PROGRAM pouS1Alarms
VAR
	idbMsgAlarm: FB_CheckMessageBounds;

END_VAR

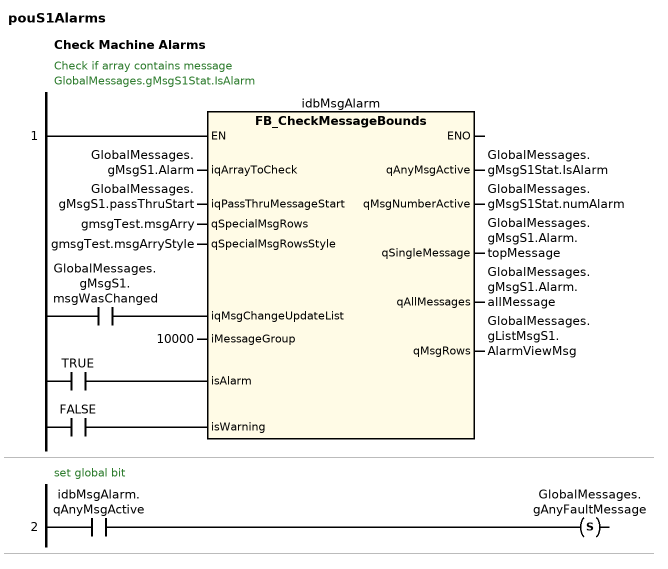
// NETWORK 1: Check Machine Alarms
// Check if array contains message
//
// GlobalMessages.gMsgS1Stat.IsAlarm
idbMsgAlarm(
    iqArrayToCheck := GlobalMessages.gMsgS1.Alarm,
    iqPassThruMessageStart := GlobalMessages.gMsgS1.passThruStart,
    qSpecialMsgRows := gmsgTest.msgArry,
    qSpecialMsgRowsStyle := gmsgTest.msgArryStyle,
    iqMsgChangeUpdateList := GlobalMessages.gMsgS1.msgWasChanged,
    iMessageGroup := 10000,
    isAlarm := TRUE,
    isWarning := FALSE,
    qAnyMsgActive => GlobalMessages.gMsgS1Stat.IsAlarm,
    qMsgNumberActive => GlobalMessages.gMsgS1Stat.numAlarm,
    qSingleMessage => GlobalMessages.gMsgS1.Alarm.topMessage,
    qAllMessages => GlobalMessages.gMsgS1.Alarm.allMessage,
    qMsgRows => GlobalMessages.gListMsgS1.AlarmViewMsg); // FB_CheckMessageBounds

// NETWORK 2
// set global bit
GlobalMessages.gAnyFaultMessage S= idbMsgAlarm.qAnyMsgActive;

END_PROGRAM

(* stored: Version 1.1.0.1, ProductVersion 3.1.4024.12
   POU pouS1Alarms: Id {4e168d6b-ccd5-440b-8127-bea095611032}, SpecialFunc None *)
